// TIA Portal V20 export
FUNCTION "Start&EndTime" : Void   // FC20224, LAD
{ S7_Optimized_Access := 'FALSE' }
// stored: AutoNumber false, SetENOAutomatically false
   VAR_INPUT
      ReadEnable : Bool;
      SelectionIndex : Int;
      DB_Source : DB_ANY;
   END_VAR
   VAR_TEMP
      i_dummy : Int;
      i_DB_Source : Int;
      i_SourceSize : Int;
      i_StartAdressSource01 : Int;
      i_StartAdressSource02 : Int;
      di_AdressSource01 : DInt;
      di_AdressSource02 : DInt;
      pa_Any01 : Any;
      pa_Any02 : Any;
      t_DTL : DTL;
      StringOfTheCurrentTime : String[32];
   END_VAR
BEGIN

NETWORK
TITLE = Read time of day
      CALL  RD_SYS_T
      ( RET_VAL := #i_dummy,
        OUT     := #t_DTL
      );


NETWORK
TITLE = DTL to string
      CALL  "DTLToString"
      ( inDTL   := #t_DTL,
        Ret_Val := #StringOfTheCurrentTime
      );


NETWORK
TITLE = Init. Variables
      OPN   #DB_Source;
      L     DBNO;
      T     #i_DB_Source;

      L     838;
      T     #i_SourceSize;
//==> StartTime
      L     250;
      T     #i_StartAdressSource01;
//==> EndTime
      L     284;
      T     #i_StartAdressSource02;


NETWORK
TITLE = Write data
      A     #ReadEnable;
      JC    Y_VI;
      JU    N_VI;
Y_VI: NOP   0;
// STRUCTURE:
// BYTE 0  : 10h       -> S7
// BYTE 1  : 13h       -> String
// BYTE 2-3: Length of data
// BYTE 4-5: DB Number
// BYTE 6  : Area 84h=DB
// BYTE 6-8: Startadress

      L     #SelectionIndex;
      L     1;
      -D;
      L     #i_SourceSize;
      *D;
      L     #i_StartAdressSource01;
      +D;
      T     #di_AdressSource01;

      L     P##pa_Any01;
      LAR1;

      L     B#16#10;
      T     LB [AR1, P#0.0];
      L     B#16#2;
      T     LB [AR1, P#1.0];
      L     32;
      T     LW [AR1, P#2.0];
      L     #i_DB_Source;
      T     LW [AR1, P#4.0];
      L     #di_AdressSource01;
      SLD   3;
      OD    DW#16#84000000;
      T     LD [AR1, P#6.0];
//==>Copty to . . .
      CALL  BLKMOV
      ( SRCBLK  := #StringOfTheCurrentTime,
        RET_VAL := #i_dummy,
        DSTBLK  := #pa_Any01
      );


      L     #SelectionIndex;
      L     1;
      -D;
      L     #i_SourceSize;
      *D;
      L     #i_StartAdressSource02;
      +D;
      T     #di_AdressSource02;

      L     P##pa_Any02;
      LAR2;

      L     B#16#10;
      T     LB [AR2, P#0.0];
      L     B#16#2;
      T     LB [AR2, P#1.0];
      L     32;
      T     LW [AR2, P#2.0];
      L     #i_DB_Source;
      T     LW [AR2, P#4.0];
      L     #di_AdressSource02;
      SLD   3;
      OD    DW#16#84000000;
      T     LD [AR2, P#6.0];

//==>Copty to . . .
      CALL  BLKMOV
      ( SRCBLK  := #StringOfTheCurrentTime,
        RET_VAL := #i_dummy,
        DSTBLK  := #pa_Any02
      );

N_VI: NOP   0;
END_FUNCTION
